PROGRAM interlocks
VAR PERSISTENT
	nv_3110_a_open: BOOL;
	alm_lt_3012_a_low: BOOL;
	intlk_u3112: BOOL;
	nv_3210_a_open: BOOL;
	nv_3310_a_open: BOOL;
	intlk_u3212: BOOL;
	intlk_u3312: BOOL;
	alm_lt_3102_a_low: BOOL;
	alm_lt_3202_a_low: BOOL;
	alm_lt_3302_a_low: BOOL;
	alm_lt_3153_a_low: BOOL;
	intlk_u3160: BOOL;
	alm_lt_3253_a_low: BOOL;
	intlk_u3260: BOOL;
	alm_lt_3353_a_low: BOOL;
	intlk_u3360: BOOL;
	nv_3372_a_open: BOOL;
	intlk_u3370: BOOL;
	alm_lt_3402_a_low: BOOL;
	nv_3135_a_open: BOOL;
	nv_3235_a_open: BOOL;
	nv_3335: BOOL;
	nv_3335_a_open: BOOL;
	intlk_nv3110: BOOL;
	u_3112_a_running: BOOL;
END_VAR

VAR
	intlk_nv3210: BOOL;
	u_3212_a_running: BOOL;
	intlk_nv3310: BOOL;
	u_3312_a_running: BOOL;
	u_3112_a_intlk: BOOL;
	nv_3110_a_intlk: BOOL;
	u_3212_a_intlk: BOOL;
	nv_3210_a_intlk: BOOL;
	u_3312_a_intlk: BOOL;
	nv_3310_a_intlk: BOOL;
	u_3160_a_intlk: BOOL;
	u_3260_a_intlk: BOOL;
	u_3360_a_intlk: BOOL;
	u_3370_a_intlk: BOOL;
	u_3405_a_intlk: BOOL;
END_VAR

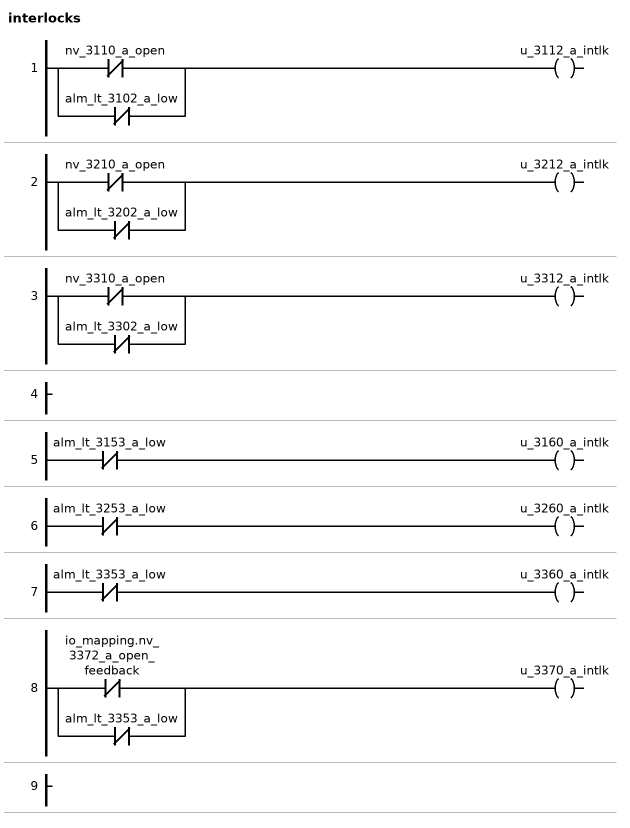
// NETWORK 1
u_3112_a_intlk := NOT nv_3110_a_open OR NOT alm_lt_3102_a_low;

// NETWORK 2
u_3212_a_intlk := NOT nv_3210_a_open OR NOT alm_lt_3202_a_low;

// NETWORK 3
u_3312_a_intlk := NOT nv_3310_a_open OR NOT alm_lt_3302_a_low;

// NETWORK 4

// NETWORK 5
u_3160_a_intlk := NOT alm_lt_3153_a_low;

// NETWORK 6
u_3260_a_intlk := NOT alm_lt_3253_a_low;

// NETWORK 7
u_3360_a_intlk := NOT alm_lt_3353_a_low;

// NETWORK 8
u_3370_a_intlk := NOT io_mapping.nv_3372_a_open_feedback OR NOT alm_lt_3353_a_low;

// NETWORK 9

END_PROGRAM

(* stored: Version 1.1.0.1, ProductVersion 3.1.4024.12
   POU interlocks: Id {5e6ac187-5fbb-479f-b495-0ce9f8a80e37}, SpecialFunc None *)
